FUNCTION_BLOCK PWMFunction
VAR_INPUT
	dutyCycle : REAL; // In % = t_ein / maxCount
	A : REAL; // Amplitude
	f : REAL; // Frequenz
	cycleTicks : REAL;
END_VAR

VAR_OUTPUT
	freqTooHigh : BOOL; //Verknüpfen mit roter LED
	pwm_Signal : REAL;
END_VAR

VAR
	T : REAL; // Zeit die das System braucht um den Funktionsblock einmal auzuführen
	fMax : REAL; // Maximale Frequnez die mit der TaskZeit erreicht werden kann
	counter : REAL;
	maxCount : REAL;
	t_ein : REAL;
END_VAR

// Taktzeit aus cycleTicks berechnen
T  := ((cycleTicks*1.0) / 1000.0);
IF T > 0.0 THEN
	fMax := 1.0 / T;
END_IF
IF f > fMax THEN
	freqTooHigh := TRUE;
	f := fMax;
END_IF
IF f > 0.0 THEN
	maxCount := (1.0 / f);
END_IF

t_ein := (dutyCycle / 100.0) * maxCount;

// Hauptzähler für Sägezahnrefernez
IF counter < maxCount THEN
	
	// PWM Generator
	IF t_ein >= counter THEN
		pwm_Signal := A;
	ELSE
		pwm_Signal := 0.0;
	END_IF
	counter := counter + T;
		
ELSIF counter >= maxCount THEN
	counter := 0.0;
END_IF

END_FUNCTION_BLOCK

(* stored: Version 1.1.0.1, ProductVersion 3.1.4022.10
   POU PWMFunction: Id {bb6bacc8-e748-4cb5-8e15-22121f2a203b}, SpecialFunc None *)
